FUNCTION_BLOCK FB_PneumaticAxis

VAR
    _stPneumaticAxis: REFERENCE TO ST_PneumaticAxisStruct;
    _iPressureGroup: I_PressureGroup;

    eState: E_PneumaticAxisState := E_PneumaticAxisState.eFailSafe;
    eSetValveState: E_PneumaticAxisValveState := eVALVE_OFF;
    eActValveState: E_PneumaticAxisValveState := eVALVE_OFF;

    apEndSwitch: ARRAY [eVALVE_OFF..eVALVE_ON] OF POINTER TO BOOL;
    apMoveTimeLimit: ARRAY [eVALVE_OFF..eVALVE_ON] OF POINTER TO INT;

    atonMoving: ARRAY [eVALVE_OFF..eVALVE_ON] OF TON;
    afElapsedTime: ARRAY [eVALVE_OFF..eVALVE_ON] OF REAL;
    afElapsedTimeTotal: ARRAY [eVALVE_OFF..eVALVE_ON] OF REAL;

    bPSSPermitNeeded: BOOL;
    bPSSPermitMissing: BOOL;
    bInterlockRequest: BOOL;

    tonInitializeTimer: TON := (PT := tINIT);
    bInitPointers: BOOL := TRUE;

    tonErrorAutoReset: TON := (PT := tAUTO_ERROR_RESET);
    rtrigReset: R_TRIG;
    artrigMoveCommand: ARRAY [eVALVE_OFF..eVALVE_ON] OF R_TRIG;
END_VAR
VAR CONSTANT
    eVALVE_OFF: E_PneumaticAxisValveState := E_PneumaticAxisValveState.eValveOff;
    eVALVE_ON: E_PneumaticAxisValveState := E_PneumaticAxisValveState.eValveOn;
    tINIT: TIME := T#3S;
    tAUTO_ERROR_RESET: TIME := T#3S;
END_VAR

PROPERTY bErrorPresent : BOOL
GET
bErrorPresent := _stPneumaticAxis.ePneumaticAxisErrors <> E_PneumaticAxisErrors.eNoError;
END_GET
END_PROPERTY

PROPERTY eError : E_PneumaticAxisErrors
GET
eError := _stPneumaticAxis.ePneumaticAxisErrors;
END_GET
SET // PRIVATE
IF eError <> E_PneumaticAxisErrors.eNoError THEN
    _stPneumaticAxis.ePneumaticAxisErrors := eError;
END_IF
END_SET
END_PROPERTY

METHOD PRIVATE EndOfCycle
_stPneumaticAxis.stPneumaticAxisControl.bInterlock := FALSE;
END_METHOD

METHOD FB_reinit : BOOL
VAR_INPUT
END_VAR
bInitPointers := TRUE;
END_METHOD

PROPERTY iPressureGroup : I_PressureGroup
GET
iPressureGroup := _iPressureGroup;
END_GET
SET
_iPressureGroup := iPressureGroup;
END_SET
END_PROPERTY

//Controls move timer and timing data
METHOD PRIVATE mControl_MoveTimer
VAR_INPUT
    eValve: E_PneumaticAxisValveState;
END_VAR
VAR
    bStart: BOOL;
END_VAR
bStart := (eState = E_PneumaticAxisState.eMoving)
    AND (eValve = eSetValveState);

//Update Time
IF atonMoving[eValve].IN THEN
    afElapsedTime[eValve] := TIME_TO_REAL(atonMoving[eValve].ET) / 1000.0;

    IF NOT bStart THEN
        afElapsedTimeTotal[eValve] := afElapsedTime[eValve];
    END_IF
END_IF

//Call
atonMoving[eValve](
    IN := bStart,
    PT := INT_TO_TIME(apMoveTimeLimit[eValve]^ * 1000));
END_METHOD

//Controls error reset
METHOD PRIVATE mControl_Reset
VAR
	bReset: BOOL := FALSE;
END_VAR
rtrigReset(CLK := _stPneumaticAxis.stPneumaticAxisControl.bReset);

tonErrorAutoReset.IN := FALSE;
  
CASE eError OF
    E_PneumaticAxisErrors.eAirPressureErrorLow:
        tonErrorAutoReset.IN := NOT _iPressureGroup.bPressureLow;
        bReset := tonErrorAutoReset.Q;
        
    E_PneumaticAxisErrors.eAirPressureErrorHigh:
        tonErrorAutoReset.IN := NOT _iPressureGroup.bPressureHigh;
        bReset := tonErrorAutoReset.Q;
        
    E_PneumaticAxisErrors.eNoPSSPermit:
        bReset := NOT bPSSPermitMissing;
        
    E_PneumaticAxisErrors.eNoSignalFromEndSwitchValveOff:
        bReset := apEndSwitch[eVALVE_OFF]^;
        
    E_PneumaticAxisErrors.eEndSwitchSignalConflict:
        bReset := NOT (apEndSwitch[eVALVE_OFF]^ 
            AND apEndSwitch[eVALVE_ON]^);
        
    E_PneumaticAxisErrors.eValveOffInterlocked,
    E_PneumaticAxisErrors.eValveOnInterlocked:
        bReset := NOT bInterlockRequest;
        
END_CASE

tonErrorAutoReset();

IF rtrigReset.Q OR bReset THEN
    _stPneumaticAxis.ePneumaticAxisErrors := E_PneumaticAxisErrors.eNoError;
END_IF
END_METHOD

//Controls set valve state 
METHOD PRIVATE mControl_SetValveState
IF eState <> E_PneumaticAxisState.eMoving THEN
    eSetValveState := eActValveState;
END_IF

//Update set valve state
IF artrigMoveCommand[eVALVE_OFF].Q 
	OR bPSSPermitMissing 
THEN
	eSetValveState := eVALVE_OFF;
ELSIF artrigMoveCommand[eVALVE_ON].Q 
    AND (eState <> E_PneumaticAxisState.eMoving)
THEN
	eSetValveState := eVALVE_ON;
END_IF
END_METHOD

//Control state change requests
METHOD mControl_State
VAR_INPUT
    eNextState: E_PneumaticAxisState;
END_VAR
//Try to set initial state to standstill on init
IF tonInitializeTimer.Q THEN
    IF apEndSwitch[eVALVE_OFF]^
        OR apEndSwitch[eVALVE_ON]^
    THEN
        eNextState := E_PneumaticAxisState.eInPosition;
    END_IF
END_IF

//Change to next state, if no error present
IF bErrorPresent
    AND (eState <> E_PneumaticAxisState.eInterlocked)
THEN
    eState := E_PneumaticAxisState.eFailSafe;
ELSE
    eState := eNextState;
END_IF
END_METHOD

METHOD PRIVATE mInit : BOOL
IF NOT __ISVALIDREF(_stPneumaticAxis) THEN
    RETURN;
END_IF

_iPressureGroup :=
    GVL.afbPressureGroup[_stPneumaticAxis.stPneumaticAxisConfig.eSelectPneumaticAxisGroup];

IF bInitPointers THEN
    apEndSwitch[eVALVE_OFF] := ADR(_stPneumaticAxis.stPneumaticAxisInputs.bEndSwitchValveOff);
    apMoveTimeLimit[eVALVE_OFF] :=
        ADR(_stPneumaticAxis.stPneumaticAxisConfig.nTimeLimitMovingWithValveOff);

    apEndSwitch[eVALVE_ON] := ADR(_stPneumaticAxis.stPneumaticAxisInputs.bEndSwitchValveOn);
    apMoveTimeLimit[eVALVE_ON] :=
        ADR(_stPneumaticAxis.stPneumaticAxisConfig.nTimeLimitMovingWithValveOn);

    bInitPointers := FALSE;
END_IF

tonInitializeTimer();
IF tonInitializeTimer.Q THEN
    tonInitializeTimer.IN := FALSE;
END_IF

mInit := NOT tonInitializeTimer.IN;
END_METHOD

//Reads input variables and transforms them into internal variables
METHOD PRIVATE mInputs
//PSS Permit
bPSSPermitNeeded := _stPneumaticAxis.stPneumaticAxisConfig.bSafetyShutter;

_stPneumaticAxis.stPneumaticAxisStatus.bPSSPermitOK := bPSSPermitNeeded
    AND _stPneumaticAxis.stPneumaticAxisInputs.bPSSPermitOK;

bPSSPermitMissing := bPSSPermitNeeded
	AND (NOT _stPneumaticAxis.stPneumaticAxisInputs.bPSSPermitOK);
	
//Interlock
bInterlockRequest := _stPneumaticAxis.stPneumaticAxisControl.bInterlock
    AND NOT _stPneumaticAxis.stPneumaticAxisconfig.bSafetyShutter;

//Move Request
artrigMoveCommand[eVALVE_OFF](CLK := _stPneumaticAxis.stPneumaticAxisControl.bValveOffManual
    OR _stPneumaticAxis.stPneumaticAxisControl.bValveOff
    OR _stPneumaticAxis.stPneumaticAxisInputs.bValveOffManualOP1
    OR _stPneumaticAxis.stPneumaticAxisInputs.bValveOffManualOP2);

artrigMoveCommand[eVALVE_ON](CLK := _stPneumaticAxis.stPneumaticAxisControl.bValveOnManual
    OR _stPneumaticAxis.stPneumaticAxisControl.bValveOn
    OR _stPneumaticAxis.stPneumaticAxisInputs.bValveOnManualOP1
    OR _stPneumaticAxis.stPneumaticAxisInputs.bValveOnManualOP2);
END_METHOD

//Monitor: End Switch
METHOD PRIVATE mMonitor_EndSwitch : E_PneumaticAxisErrors
VAR CONSTANT
    aERROR: ARRAY [eVALVE_OFF..eVALVE_ON] OF E_PneumaticAxisErrors := [
        E_PneumaticAxisErrors.eNoSignalFromEndSwitchValveOff,
        E_PneumaticAxisErrors.eNoSignalFromEndSwitchValveOn];
END_VAR
IF NOT apEndSwitch[eActValveState]^ THEN
    mMonitor_EndSwitch := aERROR[eActValveState];
ELSIF apEndSwitch[eVALVE_OFF]^ 
	AND apEndSwitch[eVALVE_ON]^
THEN
	mMonitor_EndSwitch := E_PneumaticAxisErrors.eEndSwitchSignalConflict;
END_IF

eError := mMonitor_EndSwitch;
END_METHOD

//Monitor: Interlock
METHOD PRIVATE mMonitor_InterlockMove : E_PneumaticAxisErrors
VAR CONSTANT
    aERROR: ARRAY [eVALVE_OFF..eVALVE_ON] OF E_PneumaticAxisErrors := [
        E_PneumaticAxisErrors.eValveOffInterlocked,
        E_PneumaticAxisErrors.eValveOnInterlocked];
END_VAR
IF artrigMoveCommand[eSetValveState].Q
    AND (eSetValveState <> eActValveState)
THEN
    mMonitor_InterlockMove := aERROR[eActValveState];
END_IF

eError := mMonitor_InterlockMove;
END_METHOD

//Monitor: Move Timeout & No Movement
METHOD PRIVATE mMonitor_Move : E_PneumaticAxisErrors
VAR CONSTANT
    aERROR_TIMEOUT: ARRAY [eVALVE_OFF..eVALVE_ON] OF E_PneumaticAxisErrors := [
        E_PneumaticAxisErrors.eMovingWithValveOffTimedOut,
        E_PneumaticAxisErrors.eMovingWithValveOnTimedOut];
    aERROR_NO_MOVE: ARRAY [eVALVE_OFF..eVALVE_ON] OF E_PneumaticAxisErrors := [
        E_PneumaticAxisErrors.eNotMovingWithValveOff,
        E_PneumaticAxisErrors.eNotMovingWithValveOn];
END_VAR
//Timeout
IF atonMoving[eSetValveState].Q THEN
    IF apEndSwitch[eActValveState]^ THEN
        mMonitor_Move := aERROR_NO_MOVE[eSetValveState];
    ELSE
        mMonitor_Move := aERROR_TIMEOUT[eSetValveState];
    END_IF
END_IF

eError := mMonitor_Move;
END_METHOD

//Monitor: PSS Permit
METHOD PRIVATE mMonitor_Permit : E_PneumaticAxisErrors
IF bPSSPermitMissing
	AND artrigMoveCommand[eVALVE_ON].Q
THEN
    mMonitor_Permit := E_PneumaticAxisErrors.eNoPSSPermit;
END_IF

eError := mMonitor_Permit;
END_METHOD

//Monitor: Pressure Low & High (Auto-Resets)
METHOD PRIVATE mMonitor_Pressure : E_PneumaticAxisErrors
IF _iPressureGroup.bPressureLow THEN
    mMonitor_Pressure := E_PneumaticAxisErrors.eAirPressureErrorLow;
END_IF

IF _iPressureGroup.bPressureHigh THEN
    mMonitor_Pressure := E_PneumaticAxisErrors.eAirPressureErrorHigh;
END_IF

eError := mMonitor_Pressure;
END_METHOD

//Updates the status/output variables
METHOD PRIVATE mOutputs
//Actuate Solenoids
_stPneumaticAxis.stPneumaticAxisOutputs.bSolenoid1On :=
    //EITHER: Moving with Set ValveOn
    (eState = E_PneumaticAxisState.eMoving
    AND eSetValveState = E_PneumaticAxisValveState.eValveOn)
    //OR: InPosition / Interlocked in Act ValveOn
    OR ((eState = E_PneumaticAxisState.eInPosition
    OR eState = E_PneumaticAxisState.eInterlocked)
    AND eActValveState = E_PneumaticAxisValveState.eValveOn);

_stPneumaticAxis.stPneumaticAxisOutputs.bSolenoid2On :=
    //MUST: Bistable mode
    _stPneumaticAxis.stPneumaticAxisConfig.ePneumaticAxisMode = E_PneumaticAxisMode.eBistable
    //EITHER: Moving with Set ValveOff
    AND ((eState = E_PneumaticAxisState.eMoving
    AND eSetValveState = E_PneumaticAxisValveState.eValveOff)
    //OR: InPosition / Interlocked in Act ValveOff
    OR ((eState = E_PneumaticAxisState.eInPosition
    OR eState = E_PneumaticAxisState.eInterlocked)
    AND eActValveState = E_PneumaticAxisValveState.eValveOff));

//Pressure
_stPneumaticAxis.stPneumaticAxisStatus.bAirPressureLow := _iPressureGroup.bPressureLow;
_stPneumaticAxis.stPneumaticAxisStatus.bAirPressureHigh := _iPressureGroup.bPressureHigh;

//Valve Off
_stPneumaticAxis.stPneumaticAxisStatus.bInPositionValveOff := apEndSwitch[eVALVE_OFF]^;

_stPneumaticAxis.stPneumaticAxisStatus.bMovingWithValveOff :=
    (eState = E_PneumaticAxisState.eMoving)
    AND (eSetValveState = E_PneumaticAxisValveState.eValveOff);

_stPneumaticAxis.stPneumaticAxisStatus.bTimeElapsedMovingWithValveOff := afElapsedTime[eVALVE_OFF];

_stPneumaticAxis.stPneumaticAxisStatus.bSolenoid1Active :=
    _stPneumaticAxis.stPneumaticAxisOutputs.bSolenoid1On;

//Valve On
_stPneumaticAxis.stPneumaticAxisStatus.bInPositionValveOn := apEndSwitch[eVALVE_ON]^;

_stPneumaticAxis.stPneumaticAxisStatus.bMovingWithValveOn :=
    (eState = E_PneumaticAxisState.eMoving)
    AND (eSetValveState = E_PneumaticAxisValveState.eValveOn);

_stPneumaticAxis.stPneumaticAxisStatus.fTimeElapsedMovingWithValveOn := afElapsedTime[eVALVE_ON];

_stPneumaticAxis.stPneumaticAxisStatus.bSolenoid2Active :=
    _stPneumaticAxis.stPneumaticAxisOutputs.bSolenoid2On;

//Error
_stPneumaticAxis.stPneumaticAxisStatus.bError := bErrorPresent;
END_METHOD

//Maps the current state and errors into an status info text
METHOD PRIVATE mStatusInfo
CASE _stPneumaticAxis.ePneumaticAxisErrors OF

    E_PneumaticAxisErrors.eAirPressureErrorLow:
        _stPneumaticAxis.stPneumaticAxisStatus.sStatus := 'ERROR: AIR PRESSURE TOO LOW';

    E_PneumaticAxisErrors.eAirPressureErrorHigh:
        _stPneumaticAxis.stPneumaticAxisStatus.sStatus := 'ERROR: AIR PRESSURE TOO HIGH';

    E_PneumaticAxisErrors.eNoSignalFromEndSwitchValveOff:
        _stPneumaticAxis.stPneumaticAxisStatus.sStatus := 'ERROR: NO SIGNAL FROM END SWITCH VALVE OFF';

    E_PneumaticAxisErrors.eNoSignalFromEndSwitchValveOn:
        _stPneumaticAxis.stPneumaticAxisStatus.sStatus := 'ERROR: NO SIGNAL FROM END SWITCH VALVE ON';

    E_PneumaticAxisErrors.eNotMovingWithValveOff:
        _stPneumaticAxis.stPneumaticAxisStatus.sStatus := 'ERROR: VALVE OFF NOT MOVING';

    E_PneumaticAxisErrors.eNotMovingWithValveOn:
        _stPneumaticAxis.stPneumaticAxisStatus.sStatus := 'ERROR: VALVE ON NOT MOVING';

    E_PneumaticAxisErrors.eMovingWithValveOffTimedOut:
        _stPneumaticAxis.stPneumaticAxisStatus.sStatus := 'ERROR: VALVE OFF TIMEDOUT';

    E_PneumaticAxisErrors.eMovingWithValveOnTimedOut:
        _stPneumaticAxis.stPneumaticAxisStatus.sStatus := 'ERROR: VALVE ON TIMEDOUT';

    E_PneumaticAxisErrors.eValveOffInterlocked:
        _stPneumaticAxis.stPneumaticAxisStatus.sStatus := 'ERROR: VALVE OFF INTERLOCKED';

    E_PneumaticAxisErrors.eValveOnInterlocked:
        _stPneumaticAxis.stPneumaticAxisStatus.sStatus := 'ERROR: VALVE ON INTERLOCKED';

    E_PneumaticAxisErrors.eNoError:
        CASE eState OF
            E_PneumaticAxisState.eInPosition:
                _stPneumaticAxis.stPneumaticAxisStatus.sStatus := 'NO_ERRORS_READY_TO_START';
            E_PneumaticAxisState.eMoving:
                IF eSetValveState = E_PneumaticAxisValveState.eValveOn THEN
                    _stPneumaticAxis.stPneumaticAxisStatus.sStatus := 'MOVING_WITH_VALVE_ON';
                ELSE
                    _stPneumaticAxis.stPneumaticAxisStatus.sStatus := 'MOVING_WITH_VALVE_OFF';
                END_IF
            E_PneumaticAxisState.eInterlocked:
                _stPneumaticAxis.stPneumaticAxisStatus.sStatus := 'WARNING: INTERLOCK ON, CAN NOT MOVE';
        END_CASE

    ELSE
        _stPneumaticAxis.stPneumaticAxisStatus.sStatus := 'UNKNOWN_STATE';
END_CASE
END_METHOD

METHOD PUBLIC Run
VAR
    eNextState: E_PneumaticAxisState;
END_VAR
IF NOT mInit() THEN
    RETURN;
END_IF

mInputs();

mControl_MoveTimer(eValve := eVALVE_OFF);
mControl_MoveTimer(eValve := eVALVE_ON);
mControl_SetValveState();

mMonitor_Pressure();
mMonitor_Permit();

eNextState := eState;
CASE eState OF
    E_PneumaticAxisState.eFailSafe:
        IF artrigMoveCommand[eVALVE_OFF].Q 
            OR artrigMoveCommand[eVALVE_ON].Q 
        THEN
            eNextState := E_PneumaticAxisState.eMoving;
        ELSIF apEndSwitch[eVALVE_OFF]^ THEN
            eActValveState := eVALVE_OFF;
            eNextState := E_PneumaticAxisState.eInPosition;
        END_IF

    E_PneumaticAxisState.eInPosition:
        mMonitor_EndSwitch();

        IF bInterlockRequest THEN
            eNextState := E_PneumaticAxisState.eInterlocked;
        ELSIF eSetValveState <> eActValveState THEN
            eNextState := E_PneumaticAxisState.eMoving;
        END_IF

    E_PneumaticAxisState.eMoving:
        mMonitor_Move();

        IF apEndSwitch[eSetValveState]^ THEN
            eActValveState := eSetValveState;
            eNextState := E_PneumaticAxisState.eInPosition;
        END_IF

    E_PneumaticAxisState.eInterlocked:
        mMonitor_InterlockMove();

        IF NOT bInterlockRequest THEN
            eNextState := E_PneumaticAxisState.eInPosition;
        END_IF
END_CASE

mControl_State(eNextState := eNextState);
mControl_Reset();

mStatusInfo();
mOutputs();

EndOfCycle();
END_METHOD

PROPERTY PUBLIC stPneumaticAxis : REFERENCE TO ST_PneumaticAxisStruct
GET
stPneumaticAxis REF= _stPneumaticAxis;
END_GET
SET
_stPneumaticAxis REF= stPneumaticAxis;
END_SET
END_PROPERTY

END_FUNCTION_BLOCK

(* stored: Version 1.1.0.1
   POU FB_PneumaticAxis: Id {0ba43c5d-0b1b-4802-81a2-a56c90343a83}, SpecialFunc None
   Folder Control Methods: Id {39c4bcb2-31af-075e-197a-162c75539148}
   Folder Init Methods: Id {8087fea6-af25-066c-2ec8-166e5ff52603}
   Folder Monitor Methods: Id {1de9d575-2430-0608-3cc7-4848c696c067}
   Folder Properties: Id {91a1fcf0-14fd-0997-1818-cca146c94024}
   Property bErrorPresent: Id {e61928f7-5b1b-0cb8-323f-b7787336ed0f}
   Get Get: Id {4c00db51-9bfe-0487-2f10-0681dde6f968}
   Property eError: Id {32047246-0707-0216-16bf-04057767b842}
   Get Get: Id {f3f6439d-58c8-0d64-1024-38a7f4d298fb}
   Set Set: Id {915d3ea3-4659-00d6-29b2-9f1cbc8f96f8}
   Method EndOfCycle: Id {57491fe1-9ec0-014f-336a-f4f65c1d22e5}
   Method FB_reinit: Id {1b0a7963-bcaa-0f91-0224-0925d012a176}
   Property iPressureGroup: Id {22d0755b-7b13-0cd9-272f-68eae7b24e53}
   Get Get: Id {9ea5e737-d543-0a73-2f8d-8db64b66adcb}
   Set Set: Id {c7f592e7-b27b-0c07-3f42-42fbd40d1cc1}
   Method mControl_MoveTimer: Id {b5c0d43d-0f0f-0b38-3402-746380f2c7c0}
   Method mControl_Reset: Id {eb46ca39-d8bd-0f8f-0608-612e177641a1}
   Method mControl_SetValveState: Id {22b8f3fa-139b-0f55-370c-d7d4300933e5}
   Method mControl_State: Id {5e029d34-6f19-0ae7-3102-4e3b30808b90}
   Method mInit: Id {e75835b4-a332-075c-2fc7-dc7ebd157bc6}
   Method mInputs: Id {81f9e40e-e6f9-0de7-2c11-798b5a563dc2}
   Method mMonitor_EndSwitch: Id {8fe57045-97da-0040-2f5f-3113c2e4a645}
   Method mMonitor_InterlockMove: Id {5b74e8a2-afbb-097b-0a74-e3f8f8f7ad98}
   Method mMonitor_Move: Id {759d2f8d-8e84-0713-216f-f31787094c5b}
   Method mMonitor_Permit: Id {1368e518-6934-07f8-2e25-d6a5ffa1a744}
   Method mMonitor_Pressure: Id {6586e859-2ea5-03c2-26ee-d35e5e7cbace}
   Method mOutputs: Id {e0f2114b-e095-0a99-3a69-d7ef5bca3c9b}
   Method mStatusInfo: Id {e5a09ca1-5616-0a51-3f8d-aecba84ee10e}
   Method Run: Id {4ff666c5-8aa4-4eaa-803d-5700cbef55c2}
   Property stPneumaticAxis: Id {32b385f3-2648-4c7a-b2e7-2316433a21ee}
   Get Get: Id {adb8011b-822d-0d9a-11a8-4f5c0c464fc5}
   Set Set: Id {83f042d6-81e0-4e48-8d59-f688cd15c5d1} *)
